(* IEC 61131-3 sources: ATCMcontrol_Engineering/src/TargetBase/Libs/ATCM_IEC1131_3/table_35, 2 files *)

(* ---- f_trig.st ---- *)
FUNCTION_BLOCK F_TRIG
VAR_INPUT
	CLK: BOOL;
END_VAR
VAR_OUTPUT
	Q: BOOL;
END_VAR
VAR
	M: BOOL := TRUE;
END_VAR

(*
Q := NOT CLK AND NOT M;
M := NOT CLK;
*)

inline { STDLIB(f_trig) }

END_FUNCTION_BLOCK

(* ---- r_trig.st ---- *)
FUNCTION_BLOCK R_TRIG
VAR_INPUT
	CLK: BOOL;
END_VAR
VAR_OUTPUT
	Q: BOOL;
END_VAR
VAR
	M: BOOL := FALSE;
END_VAR

(*
Q := CLK AND NOT M;
M := CLK;
*)

inline { STDLIB(r_trig) }

END_FUNCTION_BLOCK
